ABB RAPID module: Wobj_wobjnaranja.mod

MODULE Wobj_wobjnaranja
	! Points are read in order of declaration.
  ! Please do not change the order of points!

  LOCAL PERS robtarget pWobj_O_PointX1:=[[-71.3664,-648.582,653.713],[0.460308,0.58099,0.522546,-0.421323],[-2,0,-1,0],[9E+9,9E+9,9E+9,9E+9,9E+9,9E+9]];
	LOCAL PERS robtarget pWobj_O_PointX2:=[[73.0988,-647.712,658.913],[0.460311,0.580989,0.522547,-0.42132],[-1,-1,0,0],[9E+9,9E+9,9E+9,9E+9,9E+9,9E+9]];
	LOCAL PERS robtarget pWobj_O_PointY1:=[[-68.1374,-794.915,650.794],[0.460313,0.580987,0.52256,-0.421305],[-2,0,-1,0],[9E+9,9E+9,9E+9,9E+9,9E+9,9E+9]];

ENDMODULE
